FUNCTION_BLOCK MachineControlMode
VAR_INPUT
	ControlPushButtonBlock :tyPushButtonsControlBlock;	
END_VAR
VAR_OUTPUT
END_VAR
VAR
	MachineMode :tyMachineMode;
	R_TrigRunPushBotton :R_TRIG; 
	R_TrigStopPushBotton :R_TRIG; 
END_VAR

//=============================================================================
// Dmitri Raihtsaum - Copyright 2023
// Created By: Dmitri Raihtsaum
//-----------------------------------------------------------------------------
// Tested with:   Twincat 3 
// Engineering:   Twincat 3 
// Functionality: Machine controll pushbuttons logic for training
// Date: 01.04.2023
// Rev 0.1
//=============================================================================

// Mapping 
R_TrigRunPushBotton(clk:=ControlPushButtonBlock.bRunPushButton ); 
R_TrigStopPushBotton(clk:=ControlPushButtonBlock.bStopPushButton ); 
// Protection 
IF MachineMode.MashineInRunMode AND MachineMode.MashineInStopMode THEN
	MachineMode.MashineInRunMode  := FALSE; 
	MachineMode.MashineInStopMode := TRUE; 
END_IF;
IF NOT MachineMode.MashineInRunMode AND NOT  MachineMode.MashineInStopMode THEN
	MachineMode.MashineInRunMode  := FALSE; 
	MachineMode.MashineInStopMode := TRUE; 
END_IF;
// Logic 
IF R_TrigStopPushBotton.Q THEN 
	MachineMode.MashineInRunMode  := FALSE; 
	MachineMode.MashineInStopMode := TRUE  ; 
END_IF
IF R_TrigRunPushBotton.Q THEN 
	MachineMode.MashineInRunMode  := TRUE; 
	MachineMode.MashineInStopMode := FALSE ; 
END_IF
//Global Reset 
IF MachineMode.MashineInStopMode AND ControlPushButtonBlock.bResetPushButton THEN 
	GVL.bGlobalReset := TRUE;
	ELSE 
		GVL.bGlobalReset := FALSE;
END_IF;

///////////////////////END///////////////////////

END_FUNCTION_BLOCK

(* stored: Version 1.1.0.1, ProductVersion 3.1.4024.12
   POU MachineControlMode: Id {fc77a0ee-1a13-46f8-8dc6-f24d22b6fcea}, SpecialFunc None *)
